FUNCTION_BLOCK FB_Maschinentuer
VAR_INPUT
	// Sensor Eingang
	bDoorC : BOOL;
	bDoorO : BOOL;
	// Steuereingänge
	benable :BOOL; //Freigabe für Maschinenstezr
	bOpen : BOOL;
	bClose : BOOL;
END_VAR
VAR_OUTPUT
	// Aktor Ausgang
	bVentil : BOOL;
	// Zustände 
	bError : BOOL;
END_VAR
VAR
	nState : INT := 0;
END_VAR

CASE nstate OF
	0: // Tür geschlosen
		//Ausgänge setzen
		bVentil := TRUE;
		
		//Übergangsbedingung
		IF NOT bDoorc  AND benable THEN
			nstate := 3; // Tür schliesßen
		ELSIF bOpen THEN
			nstate := 1; // Tür öffnen
		END_IF
		
	1: // Tür öffnen
		// Ausgänge setzen
		bVentil := FALSE;
		
		//Übergangsbedingung
		IF bdooro THEN
			nstate := nstate + 1; // Tür geöffnet
		END_IF
		
	2: // Tür geöffnet
		bVentil := FALSE;
		
		IF bclose AND benable THEN
			nstate := 3; //Tür schließen
		END_IF
		
	3: //Tür schliesßen
		bVentil := TRUE;
		
		IF bdoorc THEN
			nstate := 0; //Tür geschlossen
		END_IF
		
END_CASE

END_FUNCTION_BLOCK

(* stored: Version 1.1.0.1, ProductVersion 3.1.4024.15
   POU FB_Maschinentuer: Id {3eac7be7-6c1d-4d83-bec9-3f5061c1c025}, SpecialFunc None *)
